// TwinCAT 3 PLC project TcUnit_Zeugwerk
// Title: TcUnit Zeugwerk
// Company: Zeugwerk GmbH
// Author: Jakob Sagatowski and Zeugwerk GmbH and contributors
// ProjectVersion: 1.3.2
// Description: TwinCAT unit testing framework. Documentation and examples are available at www.tcunit.org
// ProgramVersion: 3.1.4026.20
// libraries:
//   SysDir, * (System)
//   SysFile, * (System)
//   Tc2_Standard, * (Beckhoff Automation GmbH)
//   Tc2_System, * (Beckhoff Automation GmbH)
//   Tc2_Utilities, * (Beckhoff Automation GmbH)
//   Base Interfaces,newest,System
// project tree:
//   DUTs/ E_AssertionType.TcDUT (not stored), E_XmlError.TcDUT (not stored), ST_AdsLogStringMessage.TcDUT (not stored), ST_AssertResult.TcDUT (not stored), ST_AssertResultInstances.TcDUT (not stored), ST_AssertArrayResult.TcDUT (not stored), ST_AssertArrayResultInstances.TcDUT (not stored), ST_TestCaseResult.TcDUT (not stored), ST_TestSuiteResult.TcDUT (not stored), ST_TestSuiteResults.TcDUT (not stored), U_ExpectedOrActual.TcDUT (not stored)
//   GVLs/ GVL_Param_TcUnit.TcGVL, GVL_TcUnit.TcGVL (not stored)
//   ITFs/ I_AssertMessageFormatter.TcIO (not stored), I_TestResultLogger.TcIO (not stored), I_TestResults.TcIO (not stored)
//   POUs/ FB_AdsAssertMessageFormatter.TcPOU (not stored), FB_AdsLogStringMessageFifoQueue.TcPOU (not stored), FB_AdsTestResultLogger.TcPOU (not stored), FB_FileControl.TcPOU (not stored), FB_StreamBuffer.TcPOU (not stored), FB_XmlFileStream.TcPOU, FB_xUnitXmlPublisher.TcPOU (not stored), FB_TestResults.TcPOU (not stored), FB_AdjustAssertFailureMessageToMax253CharLength.TcPOU (not stored), FB_AssertResultStatic.TcPOU (not stored), FB_AssertArrayResultStatic.TcPOU (not stored), FB_TcUnitRunner.TcPOU (not stored), FB_Test.TcPOU (not stored), FB_TestSuite.TcPOU (not stored), FB_XmlControl.TcPOU (not stored)
//   POUs/Functions/ F_AnyToUnionValue.TcPOU (not stored), F_AnyTypeClassToString.TcPOU (not stored), F_AssertionTypeToString.TcPOU (not stored), F_GetCpuCounterAs64bit.TcPOU (not stored), F_GetTestSuiteNameFromTestInstancePath.TcPOU (not stored), F_IsAnyEqualToUnionValue.TcPOU (not stored), F_RemoveInstancePathAndProjectNameFromTestInstancePath.TcPOU (not stored), IS_TEST_FINISHED.TcPOU (not stored), RUN.TcPOU (not stored), RUN_IN_SEQUENCE.TcPOU (not stored), TCUNIT_ADSLOGSTR.TcPOU (not stored), TEST.TcPOU (not stored), TEST_FINISHED.TcPOU (not stored), TEST_FINISHED_NAMED.TcPOU (not stored), TEST_ORDERED.TcPOU (not stored)
//   POUs/Functions/WRITE_PROTECTED_/ WRITE_PROTECTED_BOOL.TcPOU (not stored), WRITE_PROTECTED_BYTE.TcPOU (not stored), WRITE_PROTECTED_DATE.TcPOU (not stored), WRITE_PROTECTED_DATE_AND_TIME.TcPOU (not stored), WRITE_PROTECTED_DINT.TcPOU (not stored), WRITE_PROTECTED_DWORD.TcPOU (not stored), WRITE_PROTECTED_INT.TcPOU (not stored), WRITE_PROTECTED_LREAL.TcPOU (not stored), WRITE_PROTECTED_REAL.TcPOU (not stored), WRITE_PROTECTED_SINT.TcPOU (not stored), WRITE_PROTECTED_STRING.TcPOU (not stored), WRITE_PROTECTED_WSTRING.TcPOU (not stored), WRITE_PROTECTED_TIME.TcPOU (not stored), WRITE_PROTECTED_TIME_OF_DAY.TcPOU (not stored), WRITE_PROTECTED_UDINT.TcPOU (not stored), WRITE_PROTECTED_UINT.TcPOU (not stored), WRITE_PROTECTED_ULINT.TcPOU (not stored), WRITE_PROTECTED_LWORD.TcPOU (not stored), WRITE_PROTECTED_LINT.TcPOU (not stored), WRITE_PROTECTED_USINT.TcPOU (not stored), WRITE_PROTECTED_WORD.TcPOU (not stored)
//   Version/ Global_Version.TcGVL

// ---- GVLs/GVL_Param_TcUnit.TcGVL
{attribute 'qualified_only'}
VAR_GLOBAL CONSTANT
    MaxNumberOfTestSuites : UINT := 1000;
    MaxNumberOfTestsForEachTestSuite : UINT := 100;
    MaxNumberOfAssertsForEachTestSuite : UINT := 1000;
    
    (* TcUnit logs complete test results. These include:
       - Number of test suites
       - Number of tests
       - Number of successful tests
       - Number of failed tests
       - Any eventual failed assertion (with the expected & actual value plus an user defined message)
       These are all printed to the ADS logger (Visual Studio error list) marked with ERROR criticality *)
    AdsLoggerEnablePublish : BOOL := TRUE;


    (* On top of the normal result, TcUnit also reports some statistics/extended information with HINT/INFO criticality.
       These statistics are more detailed results of the tests. This information is used when results are
       being collected by an external software (such as TcUnit-Runner) to do for example Jenkins integration.
       This extra information however takes time to print, so by setting the following parameter to FALSE
       it will speed up TcUnit finishing. *)
    LogExtendedResults : BOOL := FALSE;

    (* Enable (TRUE) or disable (FALSE) publishing of the xUnit Xml report *)
    xUnitEnablePublish : BOOL := TRUE;

    (* Default reserved PLC memory buffer used for composition of the xUnit xml file (64 kb default) *)
    xUnitBufferSize : UDINT := 65535;

    (* Default path and filename for the xunit testresults e.g.: for use with jenkins 

	   Use environment variables for a OS independent file path
	   - %TC_BOOTPRJPATH% -> 'C:\TwinCAT\3.1\Boot\' (Windows), '/usr/local/etc/TwinCAT/3.1/Boot/' (TC/BSD), '\Hard Disk\TwinCAT\3.1\Boot\' (Windows CE)
      - %TC_INSTALLPATH% -> 'C:\TwinCAT\3.1\' (Windows), '/usr/local/etc/TwinCAT/3.1/' (TC/BSD), '\Hard Disk\TwinCAT\3.1\' (Windows CE) *)
    xUnitFilePath : T_MaxString := '%TC_BOOTPRJPATH%tcunit_xunit_testresults.xml';

    (* This is the maximum number of ADS-messages that can be stored for reporting at the same time.
       Having a size of 2000 means that it's possible to report up to ~400 test cases in one single
       PLC cycle. Each entry consumes around 500 bytes, so with an example of a ring buffer size of
       2000 it means that TcUnit will consume around 1 MB of router memory. *) 
    AdsLogMessageFifoRingBufferSize : UINT := 2000;

    (* Time delay between a test suite is finished and the execution of the next test suite starts
       if using RUN_IN_SEQUENCE() *)
    TimeBetweenTestSuitesExecution : TIME := T#0MS;
END_VAR

// ---- Version/Global_Version.TcGVL
{attribute 'TcGenerated'}
{attribute 'no-analysis'}
{attribute 'linkalways'}
// This function has been automatically generated from the project information.
VAR_GLOBAL CONSTANT
	{attribute 'const_non_replaced'}
	stLibVersion_TcUnit_Zeugwerk : ST_LibVersion := (iMajor := 1, iMinor := 3, iBuild := 2, iRevision := 0, nFlags := 0, sVersion := '1.3.2');
END_VAR

// ---- POUs/FB_XmlFileStream.TcPOU
// This functionblock acts as a stream buffer for use with FB_XmlControl
FUNCTION_BLOCK FB_XmlFileStream EXTENDS FB_StreamBuffer
VAR
    File : FB_FileControl;
  
    BufferInitialised : BOOL := FALSE;
    Buffer : ARRAY [0..(GVL_Param_TcUnit.XUnitBufferSize - 1)] OF BYTE;  
END_VAR

// Appends a string to the buffer
PROPERTY Append : T_MaxString
SET
VAR
    ByteIn : POINTER TO BYTE;
    ByteBuffer : POINTER TO BYTE;
END_VAR
ByteIn := ADR(Append); 
ByteBuffer := _PointerToStringBuffer + _Length; // set start address

REPEAT
  
  WHILE ByteIn^ <> 0 AND _Length < _BufferSize  DO
      ByteBuffer^ := ByteIn^; //Copy the 1st byte
      _Length := _Length + 1; // set new buffer length
      ByteIn := ByteIn + 1; // calculate new start address 
      ByteBuffer := ByteBuffer + 1; // calculate new start address 
  END_WHILE;
  
  IF ByteIn^ <> 0
  THEN
    Flush();
    Clear();
    ByteBuffer := _PointerToStringBuffer;
  END_IF

UNTIL ByteIn^ = 0 END_REPEAT

ByteBuffer := _PointerToStringBuffer + _Length; // String End
ByteBuffer^ := 0; // null terminated string
END_SET
END_PROPERTY

(*
    Deletes the former file (if it exists).
    Opens the file, writes the buffer and closes it.
*)
METHOD CloseFile : SysFile.SysTypes.RTS_IEC_RESULT;
CloseFile := SysDir.CmpErrors.Errors.ERR_OK;
CloseFile := MAX(CloseFile, Flush());
CloseFile := MAX(CloseFile, File.Close());
END_METHOD

(*
    Deletes the former file (if it exists).
    Opens the file, writes the buffer and closes it.
*)
METHOD CreateFile : SysFile.SysTypes.RTS_IEC_RESULT;
CreateFile := SysDir.CmpErrors.Errors.ERR_OK;
CreateFile := MAX(CreateFile, File.Delete(Filename := GVL_Param_TcUnit.xUnitFilePath));
CreateFile := MAX(CreateFile, File.Open(Filename := GVL_Param_TcUnit.xUnitFilePath, FileAccessMode := ACCESS_MODE.AM_WRITE_PLUS));
END_METHOD

//FB_Init is always available implicitly and it is used primarily for initialization.
//The return value is not evaluated. For a specific influence, you can also declare the
//methods explicitly and provide additional code there with the standard initialization
//code. You can evaluate the return value.
METHOD FB_Init: BOOL
VAR_INPUT
    bInitRetains: BOOL; // TRUE: the retain variables are initialized (reset warm / reset cold)
    bInCopyCode: BOOL;  // TRUE: the instance will be copied to the copy code afterward (online change)   
END_VAR
SetBuffer(ADR(Buffer), GVL_Param_TcUnit.XUnitBufferSize);
END_METHOD

(*
    Deletes the former file (if it exists).
    Opens the file, writes the buffer and closes it.
*)
METHOD PRIVATE Flush : SysFile.SysTypes.RTS_IEC_RESULT;
Flush := SysDir.CmpErrors.Errors.ERR_OK;
Flush := MAX(Flush, File.Write(_PointerToStringBuffer, _Length));
Flush := MAX(Flush, File.Close());
Flush := MAX(Flush, File.Open(Filename := GVL_Param_TcUnit.xUnitFilePath, FileAccessMode := ACCESS_MODE.AM_APPEND_PLUS));
END_METHOD

END_FUNCTION_BLOCK
